PROGRAM HomingRoutine
VAR
END_VAR

CASE GVL_MOTION.HomingState OF
0:
GVL_MOTION.zCon.Execute_HOME			:= TRUE;
GVL_MOTION.HomingState					:= 1;

1:
IF GVL_MOTION.zHomeStatus.Done THEN
	GVL_MOTION.zCon.Execute_HOME		:= FALSE;
	GVL_MOTION.yCon.Execute_HOME		:= TRUE;
	GVL_MOTION.HomingState				:= 2;
END_IF

2:
IF GVL_MOTION.yHomeStatus.Done THEN
	GVL_MOTION.yCon.Execute_HOME		:= FALSE;
	GVL_MOTION.xCon.ExecuteRevUncouple	:= FALSE;
	GVL_MOTION.xCon.ExecuteUncouple 	:= FALSE;
	GVL_MOTION.xCon.ExecuteRevCouple	:= FALSE;
	//GVL_MOTION.xCon.ExecuteCouple		:= FALSE;
	GVL_MOTION.HomingState				:= 3;
END_IF

3:
IF GVL_MOTION.xOut.AxisCoupled = TRUE THEN
	GVL_MOTION.xCon.ExecuteUncouple 	:= TRUE;
END_IF
GVL_MOTION.HomingState					:= 4;

4:
GVL_MOTION.xCon.ExecuteUncouple 		:= FALSE;
GVL_MOTION.HomingState					:= 5;
	
5:
//need full cycle to set axis to couple
GVL_MOTION.RevCouplePrep				:= TRUE;
GVL_MOTION.HomingState					:= 6;

6:
GVL_MOTION.xCon.ExecuteRevCouple		:= TRUE;
GVL_MOTION.xCon.Execute_REV_HOME		:= TRUE;
GVL_MOTION.HomingState					:= 7;

7:
IF GVL_MOTION.xCHomeStatus.Done THEN
	GVL_MOTION.xCon.Execute_REV_HOME	:= FALSE;
	GVL_MOTION.xCon.ExecuteRevCouple	:= FALSE;
	GVL_MOTION.xCon.ExecuteRevUncouple	:= TRUE;		
	
	GVL_MOTION.HomingState				:= 8;
END_IF

8:
GVL_MOTION.RevCouplePrep				:= FALSE;
GVL_MOTION.HomingState					:= 9;

9:
GVL_MOTION.xCon.ExecuteRevUncouple	:= FALSE;
GVL_MOTION.xCon.ExecuteCouple		:= FALSE;
GVL_MOTION.HomingState				:= 10;

10:
GVL_MOTION.xCon.ExecuteCouple		:= TRUE;
GVL_MOTION.xCon.Execute_HOME		:= TRUE;
GVL_MOTION.HomingState				:= 11;

11:
IF GVL_MOTION.xHomeStatus.Done THEN
	GVL_MOTION.xCon.Execute_HOME		:= FALSE;
	GVL_MOTION.HomingState				:= 0;
	GVL_MOTION.HomeDone					:= TRUE;
	GVL_MOTION.EXT_CTR.CMDHOME			:= FALSE;	
END_IF


END_CASE

END_PROGRAM

(* stored: Version 1.1.0.1, ProductVersion 3.1.4026.12
   POU HomingRoutine: Id {7accc7fa-6940-4739-b56d-09b18038caf8}, SpecialFunc None *)
